// TIA Portal V16 export
// export: Created 2021-12-01T20:36:07.3309018Z, ExportSetting WithDefaults, DisplayName Totally Integrated Automation Portal, DisplayVersion V16 Update 4, DisplayName TIA Portal Version Control Interface, DisplayVersion V16 Update 2, DisplayName TIA Portal Openness, DisplayVersion V16 Update 4, DisplayName SINAMICS Startdrive Advanced, DisplayVersion V16 Update 5, DisplayName SINAMICS Startdrive G130, G150, S120, S150, SINAMICS MV, S210, DisplayVersion V16 Update 5, DisplayName SINAMICS Startdrive G110M, G120, G120C, G120D, G120P, G115D, DisplayVersion V16 Update 5, DisplayName STEP 7 Professional, DisplayVersion V16 Update 4, DisplayName STEP 7 Safety, DisplayVersion V16, DisplayName WinCC Advanced, DisplayVersion V16 Update 4
DATA_BLOCK "ST00325_SM_SA_FB_IDB"   // DB608
VERSION : 0.1
// stored: AssignedProDiagFB DIAG_PD, AutoNumber false, DBAccessibleFromOPCUA true, InstanceOfName SKID_MANAGER_SET_ATTRIBUTE_FB, InstanceOfType FB
"SKID_MANAGER_SET_ATTRIBUTE_FB"
   // VAR_INPUT
   //    PLANT_IDENTIFIER { ExternalAccessible := 'False'; ExternalVisible := 'False'; ExternalWritable := 'False'} : WString[20];
   //    SKID_NUMBER { ExternalAccessible := 'False'; ExternalVisible := 'False'; ExternalWritable := 'False'} : UDInt;
   //    SKID_ATTRIBUTE1_TYPE { ExternalAccessible := 'False'; ExternalVisible := 'False'; ExternalWritable := 'False'} : Int;
   //    SKID_ATTRIBUTE1_NAME { ExternalAccessible := 'False'; ExternalVisible := 'False'; ExternalWritable := 'False'} : String[40];
   //    SKID_ATTRIBUTE1_VALUE { ExternalAccessible := 'False'; ExternalVisible := 'False'; ExternalWritable := 'False'} : String[40];
   //    SKID_ATTRIBUTE2_TYPE { ExternalAccessible := 'False'; ExternalVisible := 'False'; ExternalWritable := 'False'} : Int;
   //    SKID_ATTRIBUTE2_NAME { ExternalAccessible := 'False'; ExternalVisible := 'False'; ExternalWritable := 'False'} : String[40];
   //    SKID_ATTRIBUTE2_VALUE { ExternalAccessible := 'False'; ExternalVisible := 'False'; ExternalWritable := 'False'} : String[40];
   //    PAYLOAD_INDEX { ExternalAccessible := 'False'; ExternalVisible := 'False'; ExternalWritable := 'False'} : UDInt;
   //    PAYLOAD_ATTRIBUTE1_TYPE { ExternalAccessible := 'False'; ExternalVisible := 'False'; ExternalWritable := 'False'} : Int;
   //    PAYLOAD_ATTRIBUTE1_NAME { ExternalAccessible := 'False'; ExternalVisible := 'False'; ExternalWritable := 'False'} : String[40];
   //    PAYLOAD_ATTRIBUTE1_VALUE { ExternalAccessible := 'False'; ExternalVisible := 'False'; ExternalWritable := 'False'} : String[40];
   //    PAYLOAD_ATTRIBUTE2_TYPE { ExternalAccessible := 'False'; ExternalVisible := 'False'; ExternalWritable := 'False'} : Int;
   //    PAYLOAD_ATTRIBUTE2_NAME { ExternalAccessible := 'False'; ExternalVisible := 'False'; ExternalWritable := 'False'} : String[40];
   //    PAYLOAD_ATTRIBUTE2_VALUE { ExternalAccessible := 'False'; ExternalVisible := 'False'; ExternalWritable := 'False'} : String[40];
   //    EXECUTE { ExternalAccessible := 'False'; ExternalVisible := 'False'; ExternalWritable := 'False'} : Bool;
   //    RESET { ExternalAccessible := 'False'; ExternalVisible := 'False'; ExternalWritable := 'False'} : Bool;
   //    TIMEOUT_SEC { ExternalAccessible := 'False'; ExternalVisible := 'False'; ExternalWritable := 'False'} : Real;
   //    HIDE_ALARM_ALL { ExternalAccessible := 'False'; ExternalVisible := 'False'; ExternalWritable := 'False'} : Bool;
   //    HIDE_ALARM_MASK { ExternalAccessible := 'False'; ExternalVisible := 'False'; ExternalWritable := 'False'} : Word;
   //    SIMULATE { ExternalAccessible := 'False'; ExternalVisible := 'False'; ExternalWritable := 'False'} : Bool;
   // END_VAR
   // VAR_OUTPUT
   //    BUSY { ExternalAccessible := 'False'; ExternalVisible := 'False'; ExternalWritable := 'False'} : Bool;
   //    DONE { ExternalAccessible := 'False'; ExternalVisible := 'False'; ExternalWritable := 'False'} : Bool;
   //    ERROR { ExternalAccessible := 'False'; ExternalVisible := 'False'; ExternalWritable := 'False'} : Bool;
   //    BYPASSED { ExternalAccessible := 'False'; ExternalVisible := 'False'; ExternalWritable := 'False'} : Bool;
   //    SIMULATED { ExternalAccessible := 'False'; ExternalVisible := 'False'; ExternalWritable := 'False'} : Bool;
   //    TIMEOUT { ExternalAccessible := 'False'; ExternalVisible := 'False'; ExternalWritable := 'False'} : Bool;
   //    EMPTY_ARGUMENTS { ExternalAccessible := 'False'; ExternalVisible := 'False'; ExternalWritable := 'False'} : Bool;
   //    STATUS_CODE { ExternalAccessible := 'False'; ExternalVisible := 'False'; ExternalWritable := 'False'} : UInt;
   // END_VAR
   // VAR_IN_OUT
   //    IF_OUT_UDT2010 : "UDT2010_SKID_ATTRIBUTE_UDT";
   //    IF_IN_UDT2100 : "UDT2100_BASE_RESPONSE_UDT";
   //    IF_HMI : "SKID_MANAGER_SET_ATTRIBUTE_HMI_UDT";
   // END_VAR
   // VAR RETAIN
   //    Alarms { ExternalAccessible := 'False'; ExternalVisible := 'False'; ExternalWritable := 'False'} : Struct
   //       EmptyArguments { ExternalAccessible := 'False'; ExternalVisible := 'False'; ExternalWritable := 'False'} : Bool;
   //       Timeout { ExternalAccessible := 'False'; ExternalVisible := 'False'; ExternalWritable := 'False'} : Bool;
   //       TransactionFailed { ExternalAccessible := 'False'; ExternalVisible := 'False'; ExternalWritable := 'False'} : Bool;
   //       Spare_3 { ExternalAccessible := 'False'; ExternalVisible := 'False'; ExternalWritable := 'False'} : Bool;
   //       Spare_4 { ExternalAccessible := 'False'; ExternalVisible := 'False'; ExternalWritable := 'False'} : Bool;
   //       Spare_5 { ExternalAccessible := 'False'; ExternalVisible := 'False'; ExternalWritable := 'False'} : Bool;
   //       Spare_6 { ExternalAccessible := 'False'; ExternalVisible := 'False'; ExternalWritable := 'False'} : Bool;
   //       Spare_7 { ExternalAccessible := 'False'; ExternalVisible := 'False'; ExternalWritable := 'False'} : Bool;
   //       Spare_8 { ExternalAccessible := 'False'; ExternalVisible := 'False'; ExternalWritable := 'False'} : Bool;
   //       Spare_9 { ExternalAccessible := 'False'; ExternalVisible := 'False'; ExternalWritable := 'False'} : Bool;
   //       Spare_10 { ExternalAccessible := 'False'; ExternalVisible := 'False'; ExternalWritable := 'False'} : Bool;
   //       Spare_11 { ExternalAccessible := 'False'; ExternalVisible := 'False'; ExternalWritable := 'False'} : Bool;
   //       Spare_12 { ExternalAccessible := 'False'; ExternalVisible := 'False'; ExternalWritable := 'False'} : Bool;
   //       Spare_13 { ExternalAccessible := 'False'; ExternalVisible := 'False'; ExternalWritable := 'False'} : Bool;
   //       Spare_14 { ExternalAccessible := 'False'; ExternalVisible := 'False'; ExternalWritable := 'False'} : Bool;
   //       Spare_15 { ExternalAccessible := 'False'; ExternalVisible := 'False'; ExternalWritable := 'False'} : Bool;
   //    END_STRUCT;
   //    HideAlarms { ExternalAccessible := 'False'; ExternalVisible := 'False'; ExternalWritable := 'False'} : Struct
   //       EmptyArguments { ExternalAccessible := 'False'; ExternalVisible := 'False'; ExternalWritable := 'False'} : Bool;
   //       Timeout { ExternalAccessible := 'False'; ExternalVisible := 'False'; ExternalWritable := 'False'} : Bool;
   //       TransactionFailed { ExternalAccessible := 'False'; ExternalVisible := 'False'; ExternalWritable := 'False'} : Bool;
   //       Spare_3 { ExternalAccessible := 'False'; ExternalVisible := 'False'; ExternalWritable := 'False'} : Bool;
   //       Spare_4 { ExternalAccessible := 'False'; ExternalVisible := 'False'; ExternalWritable := 'False'} : Bool;
   //       Spare_5 { ExternalAccessible := 'False'; ExternalVisible := 'False'; ExternalWritable := 'False'} : Bool;
   //       Spare_6 { ExternalAccessible := 'False'; ExternalVisible := 'False'; ExternalWritable := 'False'} : Bool;
   //       Spare_7 { ExternalAccessible := 'False'; ExternalVisible := 'False'; ExternalWritable := 'False'} : Bool;
   //       Spare_8 { ExternalAccessible := 'False'; ExternalVisible := 'False'; ExternalWritable := 'False'} : Bool;
   //       Spare_9 { ExternalAccessible := 'False'; ExternalVisible := 'False'; ExternalWritable := 'False'} : Bool;
   //       Spare_10 { ExternalAccessible := 'False'; ExternalVisible := 'False'; ExternalWritable := 'False'} : Bool;
   //       Spare_11 { ExternalAccessible := 'False'; ExternalVisible := 'False'; ExternalWritable := 'False'} : Bool;
   //       Spare_12 { ExternalAccessible := 'False'; ExternalVisible := 'False'; ExternalWritable := 'False'} : Bool;
   //       Spare_13 { ExternalAccessible := 'False'; ExternalVisible := 'False'; ExternalWritable := 'False'} : Bool;
   //       Spare_14 { ExternalAccessible := 'False'; ExternalVisible := 'False'; ExternalWritable := 'False'} : Bool;
   //       Spare_15 { ExternalAccessible := 'False'; ExternalVisible := 'False'; ExternalWritable := 'False'} : Bool;
   //    END_STRUCT;
   //    Instruction { ExternalAccessible := 'False'; ExternalVisible := 'False'; ExternalWritable := 'False'} : Struct
   //       Timer_Execute { ExternalAccessible := 'False'; ExternalVisible := 'False'; ExternalWritable := 'False'} : IEC_TIMER;
   //    END_STRUCT;
   //    Time_Expire { ExternalAccessible := 'False'; ExternalVisible := 'False'; ExternalWritable := 'False'} : Struct
   //       Executing { ExternalAccessible := 'False'; ExternalVisible := 'False'; ExternalWritable := 'False'} : Bool;
   //    END_STRUCT;
   //    AX { ExternalAccessible := 'False'; ExternalVisible := 'False'; ExternalWritable := 'False'} : Struct
   //       TransactionFailed { ExternalAccessible := 'False'; ExternalVisible := 'False'; ExternalWritable := 'False'} : Bool;
   //       ReadyToExecute { ExternalAccessible := 'False'; ExternalVisible := 'False'; ExternalWritable := 'False'} : Bool;
   //       Timer_Execute_PT { ExternalAccessible := 'False'; ExternalVisible := 'False'; ExternalWritable := 'False'} : DInt;
   //    END_STRUCT;
   //    Alarm_No_PD { ExternalAccessible := 'False'; ExternalVisible := 'False'; ExternalWritable := 'False'} : UInt;
   //    Warning_No_PD { ExternalAccessible := 'False'; ExternalVisible := 'False'; ExternalWritable := 'False'} : Array[0..7] of UInt;
   // END_VAR
   // VAR
   //    GLOBAL_TECUNIT_AlarmTextList_Item { ExternalAccessible := 'False'; ExternalVisible := 'False'; ExternalWritable := 'False'} : USInt;
   //    State_BypassedSkidNumber { ExternalAccessible := 'False'; ExternalVisible := 'False'; ExternalWritable := 'False'} : UDInt;
   //    AX_BypassCommandOld { ExternalAccessible := 'False'; ExternalVisible := 'False'; ExternalWritable := 'False'} : Bool;
   //    HideAlarmMesages { ExternalAccessible := 'False'; ExternalVisible := 'False'; ExternalWritable := 'False'} : Bool;
   //    ResetIndex { ExternalAccessible := 'False'; ExternalVisible := 'False'; ExternalWritable := 'False'} : Int;
   // END_VAR
BEGIN
END_DATA_BLOCK
